// TIA Portal V19 export
TYPE "lexchangetray_typeUnEmn_toRollerRecieve"
// Type: lexchangetray_typeroller_toWorkStationRollerReq
// Type: lexchangetray_typeroller_toWorkStationRollerFeedback
// stored: Access Published
   STRUCT
      feedback { S7_SetPoint := 'True'} : "lexchangetray_typeroller_toWorkStationRollerFeedback";
      req { S7_SetPoint := 'True'} : "lexchangetray_typeroller_toWorkStationRollerReq";
   END_STRUCT;
END_TYPE
